FUNCTION_BLOCK T_RemoveComponentRemovesItem EXTENDS T_UnitTestBase
VAR
END_VAR

TestFinished();

END_FUNCTION_BLOCK

(* stored: Version 1.1.0.1, ProductVersion 3.1.4024.12
   POU T_RemoveComponentRemovesItem: Id {88702719-d147-4af0-9c08-57e5b9e9e8fd}, SpecialFunc None *)
